// TIA Portal V18 export
TYPE "UDT_VirtModulesMap"
// stored: IsFailsafeCompliant false
   STRUCT
      cRack : Byte;
      cModule : Byte;
      iDiagBuffer : USInt;
      iOwnState : UInt;
   END_STRUCT;
END_TYPE
